{attribute 'qualified_only'}

VAR_GLOBAL
	nNumber : INT := 454;
END_VAR

(* stored: Version 1.1.0.1, ProductVersion 3.1.4024.16
   GVL GVL_Config: Id {9064ae18-6aa3-4688-baf7-dd118d9dd659} *)
